(* PLC project Unnamed, Unknown Unnamed 1 *)
(* stored: creationDateTime 2026-08-05T10:33:57, modificationDateTime 2026-08-05T19:04:10 *)

PROGRAM program0
  VAR
    systec_out AT %QB0.0.2.25088.1 : USINT;  (* canfestival_0/CanOpenNode_0/systec_IO-X1/0x6200-0x01: Write Outputs 0x1 to 0x8 *)
  END_VAR

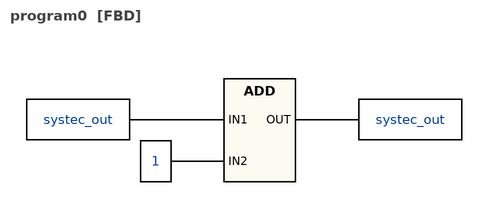
(* FBD diagram, written out as Structured Text *)
systec_out := systec_out + 1;
END_PROGRAM

CONFIGURATION config
  RESOURCE resource1 ON PLC
    TASK task0(INTERVAL := T#20ms, PRIORITY := 0);
    PROGRAM instance0 WITH task0 : program0;
  END_RESOURCE
END_CONFIGURATION
